INTERFACE I_Collection EXTENDS I_Enumerable, I_Disposable, I_EventEmitter

METHOD PUBLIC AddItem
VAR_INPUT
	Item : ANY;
END_VAR
END_METHOD

METHOD PUBLIC Clear
END_METHOD

METHOD PUBLIC Contains : BOOL;
VAR_INPUT
	Item : ANY;
END_VAR
END_METHOD

METHOD PUBLIC CopyTo : BOOL
VAR_INPUT
	Destination : ANY;
END_VAR
END_METHOD

METHOD PUBLIC CopyToLocation : BOOL
VAR_INPUT
	Destination : PVOID;
	DestinationSize : UDINT;
END_VAR
END_METHOD

PROPERTY PUBLIC Count : DINT
GET
END_GET
END_PROPERTY

METHOD PUBLIC RemoveItem : BOOL
VAR_INPUT
	Item : ANY;
END_VAR
END_METHOD

END_INTERFACE

(* stored: Version 1.1.0.1, ProductVersion 3.1.4024.12
   Itf I_Collection: Id {70b2accb-118c-42f5-8104-6faad2c2cfc3}
   Method AddItem: Id {a46b464a-5713-4157-a163-d646e3425e8a}
   Method Clear: Id {2344e2f1-4366-439e-9beb-a53fd977a5f8}
   Method Contains: Id {d98372c5-fc17-44bf-b841-3f3f44b5c96e}
   Method CopyTo: Id {eabb38d8-11ef-4981-b5dc-084a365b6ffd}
   Method CopyToLocation: Id {ca5c655f-ed6c-4dab-b806-28ef02f4713e}
   Property Count: Id {69ca6d31-a011-44c8-b83c-680b980d92f2}
   Get Get: Id {400427f4-def2-4155-af7f-13cd948a1988}
   Method RemoveItem: Id {fb9c7199-d4c2-4354-af03-01593a2b4090} *)
